FUNCTION_BLOCK StateExample IMPLEMENTS I_Statehandler
VAR
	// Interface pointer to THIS statehandler
	ipSH: I_Statehandler := THIS^;
	
	// State FBs
	fbState1: State1(ipSH);
	fbState2: State2(ipSH);

	// Interface pointer to the current state
	ipState: I_State := fbState1;
END_VAR

IF ipState <> 0 THEN
	ipState.Handle();
END_IF

METHOD SetState : BOOL
VAR_INPUT
	eNewState	: E_STATES;
END_VAR
CASE eNewState OF
	E_STATES.eState1:
		ipState := fbState1;
		
	E_STATES.eState2:
		ipState := fbState2;

	ELSE
		ADSLOGSTR(msgCtrlMask := ADSLOG_MSGTYPE_ERROR, msgFmtStr := 'unknown state', strArg := '');

END_CASE
END_METHOD

END_FUNCTION_BLOCK

(* stored: Version 1.1.0.1, ProductVersion 3.1.4024.3
   POU StateExample: Id {c5dbf8b5-3792-4102-8ec0-4477ddef9c6c}, SpecialFunc None
   Method SetState: Id {4bf7dc73-07df-4bcb-844d-3018a4efba39} *)
